{attribute addProperty BoxType "EK1122-0000-0018"}
{attribute addProperty Id "Beckhoff_ER2xxxsub_EK1100EK1100_179A0949162A_0001_ER2008_0001_0018ER2008_04E0E56B8811A_0002_ER2008_0001_0019ER2008_04E0E56B8811A_0003_ER2008_0002_0018ER2008_04E0E56B8811A_0004_ER2008_0002_0019ER2008_04E0E56B8811A_0005_ER2008_0022_0017ER2008_04E0E56B8811A_0006_ER2008_0022_0018ER2008_04E0E56B8811A_0007_ER2028_0001_0017ER2028_04E0E56B8811A_0008_ER2028_0001_0018ER2028_04E0E56B8811A_0009_ER2028_0002_0018ER2028_04E0E56B8811A_0010_ER2028_0002_0019ER2028_04E0E56B8811A_0011_ER2028_1032_0016ER2028_04E0E56B8811A_0012_ER2038_0001_0017ER2038_309488D016020A_0013_ER2038_0001_0018ER2038_309488D016020A_0014_ER2038_0002_0017ER2038_309488D016020A_0015_ER2038_0002_0018ER2038_309488D016020A_0016_ER2308_0001_0018ER2308_E58483979612A_0017_ER2308_0001_0019ER2308_E58483979612A_0018_ER2308_0002_0018ER2308_E58483979612A_0019_ER2308_0002_0019ER2308_E58483979612A_0020_ER2318_0001_0018ER2318_E58483979612A_0021_ER2318_0001_0019ER2318_E58483979612A_0022_ER2318_0002_0018ER2318_E58483979612A_0023_ER2318_0002_0019ER2318_E58483979612A_0024_ER2328_0001_0017ER2328_E58483979612A_0025_ER2328_0001_0018ER2328_E58483979612A_0026_ER2328_0002_0018ER2328_E58483979612A_0027_ER2328_0002_0019ER2328_E58483979612A_0028_ER2338_0001_0022ER2338_6598BC3916020A_0029_ER2338_0001_0023ER2338_6598BC3916020A_0030_ER2338_0002_0022ER2338_6598BC3916020A_0031_ER2338_0002_0023ER2338_6598BC3916020A_0032_ER2338_1001_0017ER2338_6598BC3916020A_0033_ER2338_1001_0018ER2338_6598BC3916020A_0034_ER2338_1002_0017ER2338_6598BC3916020A_0035_ER2338_1002_0018ER2338_6598BC3916020A_0036_ER2339_0021_0018ER2339_067D5D8B33642A_0037_ER2339_0021_0019ER2339_2F846F4A28836A_0038_ER2339_0022_0018ER2339_2F846F4A28836A_0039_ER2339_0022_0019ER2339_2F846F4A28836A_0040_ER2349_0021_0017ER2349_2F846F4A28836A_0041_ER2349_0021_0018ER2349_2F846F4A28836A_0042_ER2349_0022_0017ER2349_2F846F4A28836A_0043_ER2349_0022_0018ER2349_2F846F4A28836A_0044_ER2624_0002_0018ER2624_E7E37CC2567A_0045_ER2624_0002_0019ER2624_E7E37CC2567A_0046_ER2809_0021_0017ER2809_5A2A5F2915219A_0047_ER2809_0021_0018ER2809_5A2A5F2915219A_0048_ER2809_0022_0016ER2809_5A2A5F2915219A_0049_ER2809_0022_0017ER2809_5A2A5F2915219A_0050_ER2809_0022_0018ER2809_5A2A5F2915219"}
{attribute addProperty CRC "2314796203"}
{attribute addProperty SizeInBites "7280"}
{attribute addProperty SizeInBytes "910"}
TYPE Beckhoff_ER2xxxEK1122_89F8FCAB EXTENDS EK1122_179A0949 :
STRUCT
	{attribute addProperty Name "Beckhoff_ER2xxxsub_EK1100"}
	Beckhoff_ER2xxxsub_EK1100 : EK1100_179A0949;
	{attribute addProperty Name "A_0001_ER2008_0001_0018"}
	A_0001_ER2008_0001_0018 : ER2008_04E0E56B;
	{attribute addProperty Name "A_0002_ER2008_0001_0019"}
	A_0002_ER2008_0001_0019 : ER2008_04E0E56B;
	{attribute addProperty Name "A_0003_ER2008_0002_0018"}
	A_0003_ER2008_0002_0018 : ER2008_04E0E56B;
	{attribute addProperty Name "A_0004_ER2008_0002_0019"}
	A_0004_ER2008_0002_0019 : ER2008_04E0E56B;
	{attribute addProperty Name "A_0005_ER2008_0022_0017"}
	A_0005_ER2008_0022_0017 : ER2008_04E0E56B;
	{attribute addProperty Name "A_0006_ER2008_0022_0018"}
	A_0006_ER2008_0022_0018 : ER2008_04E0E56B;
	{attribute addProperty Name "A_0007_ER2028_0001_0017"}
	A_0007_ER2028_0001_0017 : ER2028_04E0E56B;
	{attribute addProperty Name "A_0008_ER2028_0001_0018"}
	A_0008_ER2028_0001_0018 : ER2028_04E0E56B;
	{attribute addProperty Name "A_0009_ER2028_0002_0018"}
	A_0009_ER2028_0002_0018 : ER2028_04E0E56B;
	{attribute addProperty Name "A_0010_ER2028_0002_0019"}
	A_0010_ER2028_0002_0019 : ER2028_04E0E56B;
	{attribute addProperty Name "A_0011_ER2028_1032_0016"}
	A_0011_ER2028_1032_0016 : ER2028_04E0E56B;
	{attribute addProperty Name "A_0012_ER2038_0001_0017"}
	A_0012_ER2038_0001_0017 : ER2038_309488D0;
	{attribute addProperty Name "A_0013_ER2038_0001_0018"}
	A_0013_ER2038_0001_0018 : ER2038_309488D0;
	{attribute addProperty Name "A_0014_ER2038_0002_0017"}
	A_0014_ER2038_0002_0017 : ER2038_309488D0;
	{attribute addProperty Name "A_0015_ER2038_0002_0018"}
	A_0015_ER2038_0002_0018 : ER2038_309488D0;
	{attribute addProperty Name "A_0016_ER2308_0001_0018"}
	A_0016_ER2308_0001_0018 : ER2308_E5848397;
	{attribute addProperty Name "A_0017_ER2308_0001_0019"}
	A_0017_ER2308_0001_0019 : ER2308_E5848397;
	{attribute addProperty Name "A_0018_ER2308_0002_0018"}
	A_0018_ER2308_0002_0018 : ER2308_E5848397;
	{attribute addProperty Name "A_0019_ER2308_0002_0019"}
	A_0019_ER2308_0002_0019 : ER2308_E5848397;
	{attribute addProperty Name "A_0020_ER2318_0001_0018"}
	A_0020_ER2318_0001_0018 : ER2318_E5848397;
	{attribute addProperty Name "A_0021_ER2318_0001_0019"}
	A_0021_ER2318_0001_0019 : ER2318_E5848397;
	{attribute addProperty Name "A_0022_ER2318_0002_0018"}
	A_0022_ER2318_0002_0018 : ER2318_E5848397;
	{attribute addProperty Name "A_0023_ER2318_0002_0019"}
	A_0023_ER2318_0002_0019 : ER2318_E5848397;
	{attribute addProperty Name "A_0024_ER2328_0001_0017"}
	A_0024_ER2328_0001_0017 : ER2328_E5848397;
	{attribute addProperty Name "A_0025_ER2328_0001_0018"}
	A_0025_ER2328_0001_0018 : ER2328_E5848397;
	{attribute addProperty Name "A_0026_ER2328_0002_0018"}
	A_0026_ER2328_0002_0018 : ER2328_E5848397;
	{attribute addProperty Name "A_0027_ER2328_0002_0019"}
	A_0027_ER2328_0002_0019 : ER2328_E5848397;
	{attribute addProperty Name "A_0028_ER2338_0001_0022"}
	A_0028_ER2338_0001_0022 : ER2338_6598BC39;
	{attribute addProperty Name "A_0029_ER2338_0001_0023"}
	A_0029_ER2338_0001_0023 : ER2338_6598BC39;
	{attribute addProperty Name "A_0030_ER2338_0002_0022"}
	A_0030_ER2338_0002_0022 : ER2338_6598BC39;
	{attribute addProperty Name "A_0031_ER2338_0002_0023"}
	A_0031_ER2338_0002_0023 : ER2338_6598BC39;
	{attribute addProperty Name "A_0032_ER2338_1001_0017"}
	A_0032_ER2338_1001_0017 : ER2338_6598BC39;
	{attribute addProperty Name "A_0033_ER2338_1001_0018"}
	A_0033_ER2338_1001_0018 : ER2338_6598BC39;
	{attribute addProperty Name "A_0034_ER2338_1002_0017"}
	A_0034_ER2338_1002_0017 : ER2338_6598BC39;
	{attribute addProperty Name "A_0035_ER2338_1002_0018"}
	A_0035_ER2338_1002_0018 : ER2338_6598BC39;
	{attribute addProperty Name "A_0036_ER2339_0021_0018"}
	A_0036_ER2339_0021_0018 : ER2339_067D5D8B;
	{attribute addProperty Name "A_0037_ER2339_0021_0019"}
	A_0037_ER2339_0021_0019 : ER2339_2F846F4A;
	{attribute addProperty Name "A_0038_ER2339_0022_0018"}
	A_0038_ER2339_0022_0018 : ER2339_2F846F4A;
	{attribute addProperty Name "A_0039_ER2339_0022_0019"}
	A_0039_ER2339_0022_0019 : ER2339_2F846F4A;
	{attribute addProperty Name "A_0040_ER2349_0021_0017"}
	A_0040_ER2349_0021_0017 : ER2349_2F846F4A;
	{attribute addProperty Name "A_0041_ER2349_0021_0018"}
	A_0041_ER2349_0021_0018 : ER2349_2F846F4A;
	{attribute addProperty Name "A_0042_ER2349_0022_0017"}
	A_0042_ER2349_0022_0017 : ER2349_2F846F4A;
	{attribute addProperty Name "A_0043_ER2349_0022_0018"}
	A_0043_ER2349_0022_0018 : ER2349_2F846F4A;
	{attribute addProperty Name "A_0044_ER2624_0002_0018"}
	A_0044_ER2624_0002_0018 : ER2624_E7E37CC2;
	{attribute addProperty Name "A_0045_ER2624_0002_0019"}
	A_0045_ER2624_0002_0019 : ER2624_E7E37CC2;
	{attribute addProperty Name "A_0046_ER2809_0021_0017"}
	A_0046_ER2809_0021_0017 : ER2809_5A2A5F29;
	{attribute addProperty Name "A_0047_ER2809_0021_0018"}
	A_0047_ER2809_0021_0018 : ER2809_5A2A5F29;
	{attribute addProperty Name "A_0048_ER2809_0022_0016"}
	A_0048_ER2809_0022_0016 : ER2809_5A2A5F29;
	{attribute addProperty Name "A_0049_ER2809_0022_0017"}
	A_0049_ER2809_0022_0017 : ER2809_5A2A5F29;
	{attribute addProperty Name "A_0050_ER2809_0022_0018"}
	A_0050_ER2809_0022_0018 : ER2809_5A2A5F29;
END_STRUCT
END_TYPE

(* stored: Version 1.2.0.0, ProductVersion 3.1.4024.9
   DUT Beckhoff_ER2xxxEK1122_89F8FCAB: Id {d8a872e5-98b1-4d84-8e8c-86961fdc2835} *)
